// TIA Portal V21 export
DATA_BLOCK "C0_DATA"   // DB10
{ S7_Optimized_Access := 'TRUE' }
// stored: MemoryReserve 100
   VAR
      C0 : "TypeC0";   // Copy of the current cabinet configuration
   END_VAR
BEGIN
END_DATA_BLOCK
